// TIA Portal V17 export
// export: Created 2022-02-03T14:45:13.5267827Z, ExportSetting WithDefaults, DisplayName Totally Integrated Automation Portal, DisplayVersion V17, DisplayName TIA Portal Openness, DisplayVersion V17, DisplayName TIA Portal Version Control Interface, DisplayVersion V17, DisplayName SINAMICS Startdrive Advanced, DisplayVersion V17, DisplayName SINAMICS Startdrive G130, G150, S120, S150, SINAMICS MV, S210, DisplayVersion V17, DisplayName SINAMICS Startdrive G110M, G120, G120C, G120D, G120P, G115D, DisplayVersion V17, DisplayName STEP 7 Professional, DisplayVersion V17, DisplayName STEP 7 Safety, DisplayVersion V17, DisplayName WinCC Advanced, DisplayVersion V17
DATA_BLOCK "Statistic_DB"   // DB8
VERSION : 0.1
// stored: Access Unpublished, AutoNumber true, DBAccessibleFromOPCUA true, DBAccessibleFromWebserver true, InstanceOfName Statistic, InstanceOfType FB
"Statistic"
   // VAR_INPUT
   //    Operation : Bool;
   //    occupiedBay : Array["FIRSTBAY".."LASTBAY"] of Bool;
   // END_VAR
   // VAR_IN_OUT
   //    statistics : "typeStatistics";
   // END_VAR
   // VAR
   //    statOldOperation : Bool;
   // END_VAR
   // VAR RETAIN
   //    InstIEC_Counter1 { S7_SetPoint := 'True'} : CTU_UINT;
   //    InstIEC_Counter2 { S7_SetPoint := 'True'} : CTU_UINT;
   //    INSTIEC_Counter3 { S7_SetPoint := 'True'} : CTU_UINT;
   // END_VAR
BEGIN
END_DATA_BLOCK
